FUNCTION_BLOCK FB_Stromzaehler
VAR_INPUT
	Telegramm	: ARRAY[1..cMBUS_MaxTelegrams] OF ST_MBus_Data2;

END_VAR
VAR_IN_OUT
	Zustand		: ST_SZ_Zustand;
END_VAR
VAR
END_VAR
VAR // added by the converter: edge detectors and wires of the graphical bodies
    _w1, _w2, _w3 : ANY;
END_VAR

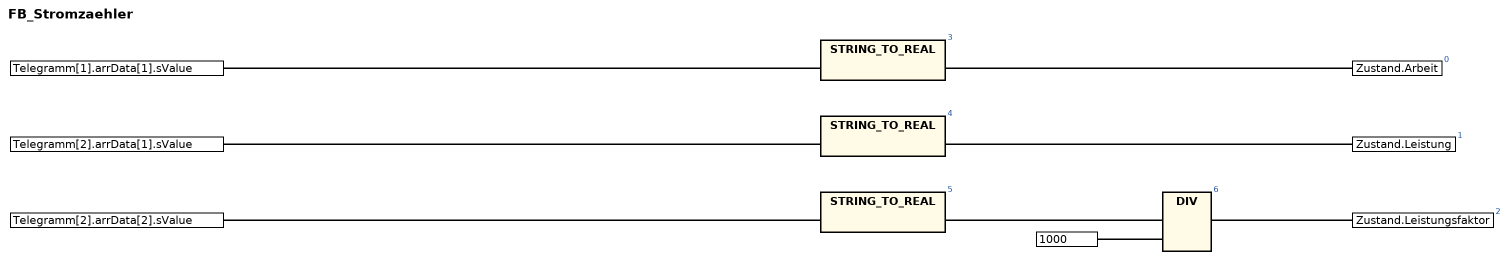
Zustand.Arbeit := _w1;
Zustand.Leistung := _w2;
Zustand.Leistungsfaktor := _w3;
_w1 := STRING_TO_REAL(Telegramm[1].arrData[1].sValue);
_w2 := STRING_TO_REAL(Telegramm[2].arrData[1].sValue);
_w3 := STRING_TO_REAL(Telegramm[2].arrData[2].sValue) / 1000;

END_FUNCTION_BLOCK

(* stored: Version 1.1.0.1, ProductVersion 3.1.4024.9
   POU FB_Stromzaehler: Id {8990275b-a658-4764-8d66-16bed02a229c}, SpecialFunc None *)
